# EPICS substitutions: jawsApp/Db/split_jaws_header_vertical.substitutions
# Creates a .db file for the header and individual vertical blades of a split full set of jaws
# This is needed where vertical and horizontal blades are controlled by separate motor IOCs and thus need to have their .dbs loaded separately.
# Expects split_jaws_horizontal.db to be loaded to work correctly

file "$(JAWS)/jawsApp/Db/jawsheader.template" {
    { P=\$(P), JAWS=\$(JAWS), mXN=\$(mXN), mXS=\$(mXS), mXE=\$(mXE), mXW=\$(mXW), ASG=\$(ASG=DEFAULT) }
}

file "$(JAWS)/jawsApp/Db/slits.template" {
    { P=\$(P), SLIT=\$(JAWS), M1=\$(mXN), M2=\$(mXS), S1=JN, S2=JS, D1=North, D2=South, GAP=VGAP, DGAP=Vertical, CENTRE=VCENT, DCENTRE=Vertical, ASG=\$(ASG=DEFAULT), EGU=\$(EGU=), CENT_DISP=\$(CENT_DISP=0) }
}

file "$(UTILITIES)/utilitiesApp/db/field_setter.template" {
    {P=\$(P), TO=\$(JAWS)JN, FROM=\$(mXN), FIELD=ADEL}
    {P=\$(P), TO=\$(JAWS)JS, FROM=\$(mXS), FIELD=ADEL}

    {P=\$(P), TO=\$(JAWS)VGAP, FROM=\$(mXN), FIELD=ADEL}

    {P=\$(P), TO=\$(JAWS)VCENT, FROM=\$(mXN), FIELD=ADEL}

}
